# EPICS autosave request: ADURL/iocs/urlIOC/iocBoot/iocURLDriver/auto_settings.req
file "URLDriver_settings.req",      P=$(P),  R=cam1:
file "ADBase_settings.req",         P=$(P),  R=cam1:
file "NDPluginBase_settings.req",   P=$(P),  R=image1:
file "NDStdArrays_settings.req",    P=$(P),  R=image1:
file "commonPlugin_settings.req",   P=$(P)
